{attribute 'linkalways'} 
{attribute 'no_explicit_call' := 'This FB is a CLASS and must be accessed using methods or properties'}
{attribute 'enable_dynamic_creation'}
FUNCTION_BLOCK MockEnumDatatype_E_TcEventClass EXTENDS EnumDatatypeBase
VAR
	localData : E_TcEventClass;
	activeData : REFERENCE TO E_TcEventClass;
	enumBaseDatatype : _UINT(localData);
END_VAR

METHOD PRIVATE AddLocalEnumeration
VAR_INPUT
	Enumeration : T_MAXSTRING;
	Value : E_TcEventClass;
END_VAR
AddEnumeration(Enumeration, Value);
END_METHOD

PROPERTY PUBLIC Address : PVOID
GET
Address := ADR(activeData);
END_GET
END_PROPERTY

METHOD PUBLIC ClearReference
VAR_INPUT
END_VAR
activeData REF= localData;
SetBaseDatatypeReference();
END_METHOD

METHOD PUBLIC Clone : I_Datatype
VAR
    pClone : POINTER TO MockEnumDatatype_E_TcEventClass;
END_VAR
pClone := __NEW(MockEnumDatatype_E_TcEventClass(InitialValue := Value));
Clone := pClone^;
END_METHOD

METHOD FB_init : BOOL
VAR_INPUT
	bInitRetains : BOOL; // if TRUE, the retain variables are initialized (warm start / cold start)
	bInCopyCode : BOOL;  // if TRUE, the instance afterwards gets moved into the copy code (online change)
	InitialValue : E_TcEventClass;
END_VAR
localData := InitialValue;
AddBaseDatatype(enumBaseDatatype);
ClearReference();

AddLocalEnumeration('TCEVENTCLASS_NONE', E_TcEventClass.TCEVENTCLASS_NONE);
AddLocalEnumeration('TCEVENTCLASS_MAINTENANCE', E_TcEventClass.TCEVENTCLASS_MAINTENANCE);
AddLocalEnumeration('TCEVENTCLASS_MESSAGE', E_TcEventClass.TCEVENTCLASS_MESSAGE);
AddLocalEnumeration('TCEVENTCLASS_HINT', E_TcEventClass.TCEVENTCLASS_HINT);
AddLocalEnumeration('TCEVENTCLASS_STATEINFO', E_TcEventClass.TCEVENTCLASS_STATEINFO);
AddLocalEnumeration('TCEVENTCLASS_INSTRUCTION', E_TcEventClass.TCEVENTCLASS_INSTRUCTION);
AddLocalEnumeration('TCEVENTCLASS_WARNING', E_TcEventClass.TCEVENTCLASS_WARNING);
AddLocalEnumeration('TCEVENTCLASS_ALARM', E_TcEventClass.TCEVENTCLASS_ALARM);
AddLocalEnumeration('TCEVENTCLASS_PARAMERROR', E_TcEventClass.TCEVENTCLASS_PARAMERROR);
END_METHOD

PROPERTY PUBLIC Identifier : T_MAXSTRING
GET
Identifier := 'E_TcEventClass';
END_GET
END_PROPERTY

METHOD IsEnumeratorValueEqual : BOOL
VAR_INPUT
	Enumerator : I_KeyValueForwardEnumerator;
END_VAR
VAR
	storedValue : E_TcEventClass;
END_VAR
IF NOT Enumerator.TryGet(storedValue) THEN
	RETURN;
END_IF

IsEnumeratorValueEqual := storedValue = activeData;
END_METHOD

METHOD PUBLIC MakeReferenceTo
VAR_INPUT
	ReferenceTarget : REFERENCE TO E_TcEventClass;
END_VAR
activeData REF= ReferenceTarget;
SetBaseDatatypeReference();
END_METHOD

METHOD PROTECTED SetBaseDatatypeReference
VAR_INPUT
END_VAR
enumBaseDatatype.MakeReferenceTo(activeData);
END_METHOD

PROPERTY PUBLIC Size : UDINT
GET
Size := SIZEOF(activeData);
END_GET
END_PROPERTY

METHOD TryMakeReferenceTo : BOOL
VAR_INPUT
	Target : I_Datatype;
END_VAR
VAR
	pTargetData : POINTER TO E_TcEventClass;
END_VAR
IF NOT IsEquivalentTo(Target) THEN
	RETURN;
END_IF

pTargetData := Target.Address;
activeData REF= pTargetData^;
SetBaseDatatypeReference();
TryMakeReferenceTo := TRUE;
END_METHOD

PROPERTY PUBLIC Value : REFERENCE TO E_TcEventClass
GET
Value REF= activeData;
END_GET
END_PROPERTY

END_FUNCTION_BLOCK

(* stored: Version 1.1.0.1, ProductVersion 3.1.4024.13
   POU MockEnumDatatype_E_TcEventClass: Id {ed11c15f-080b-47b0-9c16-bfcb6c22e48f}, SpecialFunc None
   Folder Constructor: Id {c437d3bf-99c8-4bb6-ba5c-f57d3664a913}
   Folder Private: Id {40b6a8bc-0c77-4989-b6c8-fddfa41d0501}
   Folder Protected: Id {a60a3be0-a365-4ec9-a7a1-eeb495e8fd19}
   Method AddLocalEnumeration: Id {e41f12d6-ff20-4bff-a430-34d9aeb4e5c5}
   Property Address: Id {6ad5ee74-7a7a-4ae3-865a-057a3545e8db}
   Get Get: Id {d092b0a0-6827-4d46-8013-6d4f791064c7}
   Method ClearReference: Id {cde49f5e-c099-4ba9-aa91-833cc9c39501}
   Method Clone: Id {c1240e84-ce6c-4b59-8f06-51e72af39a80}
   Method FB_init: Id {3809ebef-b7c8-4f44-8a60-871f5edbdc0e}
   Property Identifier: Id {e5b2124b-ba06-4a8e-bc86-e99b219009fb}
   Get Get: Id {e00cad37-7f14-40ad-a843-16c10c1943ca}
   Method IsEnumeratorValueEqual: Id {dc910677-5aec-4832-9fc7-3d8cd2238ef3}
   Method MakeReferenceTo: Id {d29f8781-852b-45b0-a168-a65a476b42d4}
   Method SetBaseDatatypeReference: Id {a5fa24a7-3094-4422-95b7-298d29422a4d}
   Property Size: Id {e102b3c0-651d-4a65-9198-d35311ef1bf5}
   Get Get: Id {246c0011-8a97-43f5-9eb5-42cbdc169e4f}
   Method TryMakeReferenceTo: Id {78afb75b-70bb-4e2a-97ca-f68a821d53c9}
   Property Value: Id {0814ed9d-e210-4e22-b882-ede7682b0166}
   Get Get: Id {e01c3b1b-0e4b-4d0e-a266-bff0d4b9a91a} *)
